// TIA Portal V17 export
// export: Created 2023-04-11T09:33:31.2855493Z, ExportSetting WithDefaults, DisplayName Totally Integrated Automation Portal, DisplayVersion V17 Update 3, DisplayName TIA Portal Openness, DisplayVersion V17 Update 3, DisplayName TIA Portal Version Control Interface, DisplayVersion V17, DisplayName SINAMICS Startdrive Advanced, DisplayVersion V17 Update2, DisplayName SINAMICS Startdrive G130, G150, S120, S150, SINAMICS MV, S210, DisplayVersion V17 Update2, DisplayName SINAMICS Startdrive G110M, G120, G120C, G120D, G120P, G115D, DisplayVersion V17 Update2, DisplayName STEP 7 Professional, DisplayVersion V17 Update 3, DisplayName STEP 7 Safety, DisplayVersion V17, DisplayName WinCC UA Professional, DisplayVersion V17 Update 3
FUNCTION "FC_alignStepName" : Void   // FC20, LAD
{ S7_Optimized_Access := 'TRUE' }
VERSION : 0.1
// stored: AutoNumber true, IsIECCheckEnabled false, SetENOAutomatically false, UDAEnableTagReadback false
   VAR_INPUT
      in_array : Array[0..3] of String;
      language : Int;
   END_VAR
   VAR_OUTPUT
      out_array : Array[0..3] of String;
   END_VAR
   VAR_TEMP
      i_in : Int;
      i_out : Int;
      length : Int;
   END_VAR
   VAR CONSTANT
      MAX : Int := 3;
   END_VAR
BEGIN

REGION Network 1 (SCL)
   FOR #i_out := 0 TO #MAX DO
       #out_array[#i_out] := '';
   END_FOR;

   #i_out := 0;
   FOR #i_in := 0 TO #MAX DO
       #length := LEN("DB_S1_hmi".StepsTool1[#i_in]);
       IF (#length > 0) THEN
           #out_array[#i_out] := #in_array[#i_in];
           #i_out := #i_out + 1;
       END_IF;
   END_FOR;
END_REGION
END_FUNCTION
